# EPICS substitutions: synApps_6_1/support/motor-R7-1/modules/motorOmsAsyn/iocs/omsAsynIOC/iocBoot/iocOmsAsyn/MAXv.substitutions
file "$(MOTOR)/db/asyn_motor.db"
{
pattern
{P,         N,        M,        DTYP,   PORT,  ADDR,         DESC,  EGU,  DIR,  VELO,  VBAS,  ACCL,  BDST,  BVEL,  BACC,  MRES,   PREC,  DHLM,  DLLM,  INIT}
{omsAsyn:,  1,  "m$(N)",  "asynMotor", MAXv0,    0,  "motor $(N)",  deg,  Pos,    10,     0,    .2,     0,     1,     2,  0.01,      5,     0,     0,    ""}
}
